(* Logix 5000 project; controller Turck_IOLink_All_Full_AOIs_V0_1 vendor 1 type 14 code 176 rev 32.11; software revision 32.00; part 3 of 7 *)
(* tags used below, declared in another part *)
   TBEN_I_DATA : INT[173];   // Input Data from IO Block
   TBEN_O_DATA : INT[131];   // Output Data to IO Block
   TBEN_C_DATA : SINT[160];
   DXP1_OUT : BOOL;
   DXP3_OUT : BOOL;
   DXP5_OUT : BOOL;
   DXP7_OUT : BOOL;
   IOLDevice_PORT1 : BOOL;
   IOLDevice_PORT2 : BOOL;
   IOLDevice_PORT3 : BOOL;
   IOLDevice_PORT4 : BOOL;
   IOLDevice_PORT5 : BOOL;
   IOLDevice_PORT6 : BOOL;
   IOLDevice_PORT7 : BOOL;
   IOLDevice_PORT8 : BOOL;
   DXP7_IN : BOOL;
   IOL8_DI : BOOL;
   IOL10_DI : BOOL;
   IOL12_DI : BOOL;
   IOL14_DI : BOOL;
   PORT1_Mode_IOL_or_DI : BOOL;   // 0: IO-LINK without validation 1: Port is set to DI (Power Cycle or Module Inhibit cycle require)
   PORT2_Mode_IOL_or_DI : BOOL;   // 0: IO-LINK without validation 1: Port is set to DI (Power Cycle or Module Inhibit cycle require)
   PORT3_Mode_IOL_or_DI : BOOL;   // 0: IO-LINK without validation 1: Port is set to DI (Power Cycle or Module Inhibit cycle require)
   PORT4_Mode_IOL_or_DI : BOOL;   // 0: IO-LINK without validation 1: Port is set to DI (Power Cycle or Module Inhibit cycle require)
   PORT5_Mode_IOL_or_DI : BOOL;   // 0: IO-LINK without validation 1: Port is set to DI (Power Cycle or Module Inhibit cycle require)
   PORT6_Mode_IOL_or_DI : BOOL;   // 0: IO-LINK without validation 1: Port is set to DI (Power Cycle or Module Inhibit cycle require)
   PORT7_Mode_IOL_or_DI : BOOL;   // 0: IO-LINK without validation 1: Port is set to DI (Power Cycle or Module Inhibit cycle require)
   PORT8_Mode_IOL_or_DI : BOOL;   // 0: IO-LINK without validation 1: Port is set to DI (Power Cycle or Module Inhibit cycle require)
   DisableOutput_DXP1 : BOOL;
   DisableOutput_DXP3 : BOOL;
   DisableOutput_DXP5 : BOOL;
   DisableOutput_DXP7 : BOOL;
   IOLReadActive : BOOL;
   IOLWriteActive : BOOL;
   IOL_READ_Request : BOOL;
   IOL_WRITE_Request : BOOL;
(* TBEN_Lx_8IOL_AOI, continued *)

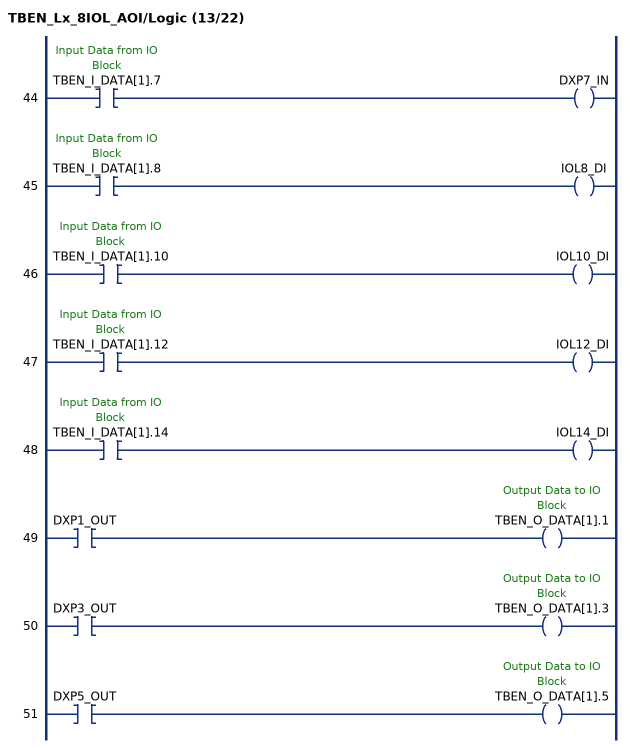
   44: XIC(TBEN_I_DATA[1].7)OTE(DXP7_IN);
   45: XIC(TBEN_I_DATA[1].8)OTE(IOL8_DI);
   46: XIC(TBEN_I_DATA[1].10)OTE(IOL10_DI);
   47: XIC(TBEN_I_DATA[1].12)OTE(IOL12_DI);
   48: XIC(TBEN_I_DATA[1].14)OTE(IOL14_DI);
   49: XIC(DXP1_OUT)OTE(TBEN_O_DATA[1].1);
   50: XIC(DXP3_OUT)OTE(TBEN_O_DATA[1].3);
   51: XIC(DXP5_OUT)OTE(TBEN_O_DATA[1].5);
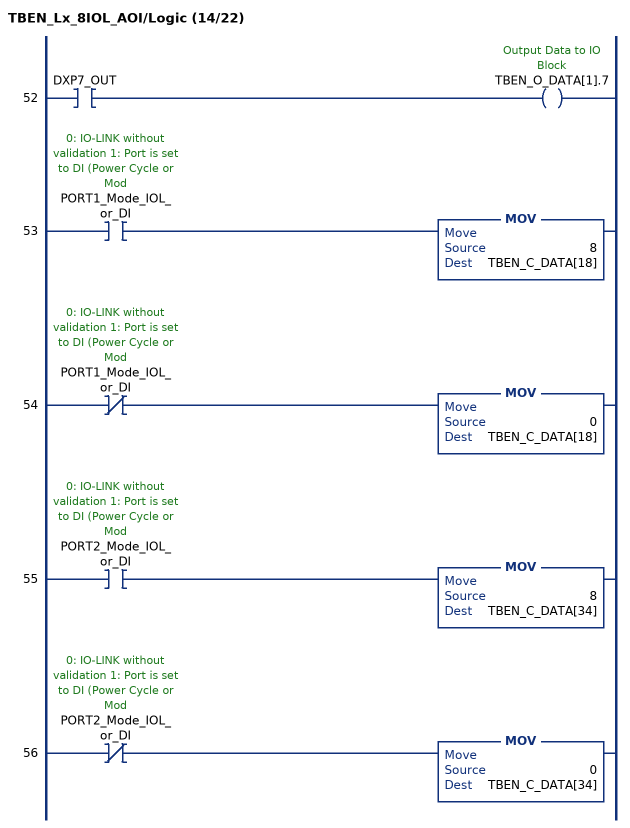
   52: XIC(DXP7_OUT)OTE(TBEN_O_DATA[1].7);
   53: XIC(PORT1_Mode_IOL_or_DI)MOV(8,TBEN_C_DATA[18]);
   54: XIO(PORT1_Mode_IOL_or_DI)MOV(0,TBEN_C_DATA[18]);
   55: XIC(PORT2_Mode_IOL_or_DI)MOV(8,TBEN_C_DATA[34]);
   56: XIO(PORT2_Mode_IOL_or_DI)MOV(0,TBEN_C_DATA[34]);
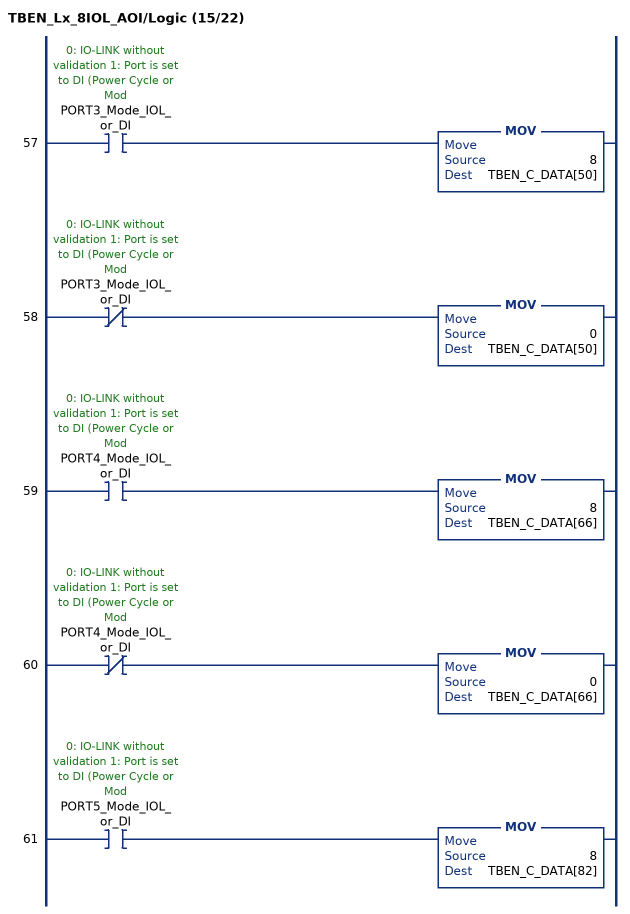
   57: XIC(PORT3_Mode_IOL_or_DI)MOV(8,TBEN_C_DATA[50]);
   58: XIO(PORT3_Mode_IOL_or_DI)MOV(0,TBEN_C_DATA[50]);
   59: XIC(PORT4_Mode_IOL_or_DI)MOV(8,TBEN_C_DATA[66]);
   60: XIO(PORT4_Mode_IOL_or_DI)MOV(0,TBEN_C_DATA[66]);
   61: XIC(PORT5_Mode_IOL_or_DI)MOV(8,TBEN_C_DATA[82]);
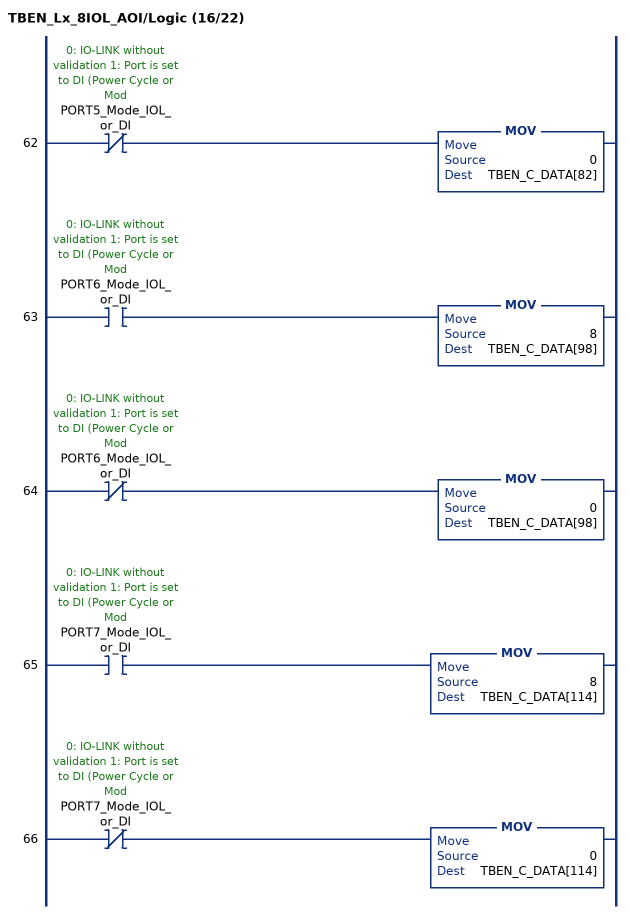
   62: XIO(PORT5_Mode_IOL_or_DI)MOV(0,TBEN_C_DATA[82]);
   63: XIC(PORT6_Mode_IOL_or_DI)MOV(8,TBEN_C_DATA[98]);
   64: XIO(PORT6_Mode_IOL_or_DI)MOV(0,TBEN_C_DATA[98]);
   65: XIC(PORT7_Mode_IOL_or_DI)MOV(8,TBEN_C_DATA[114]);
   66: XIO(PORT7_Mode_IOL_or_DI)MOV(0,TBEN_C_DATA[114]);
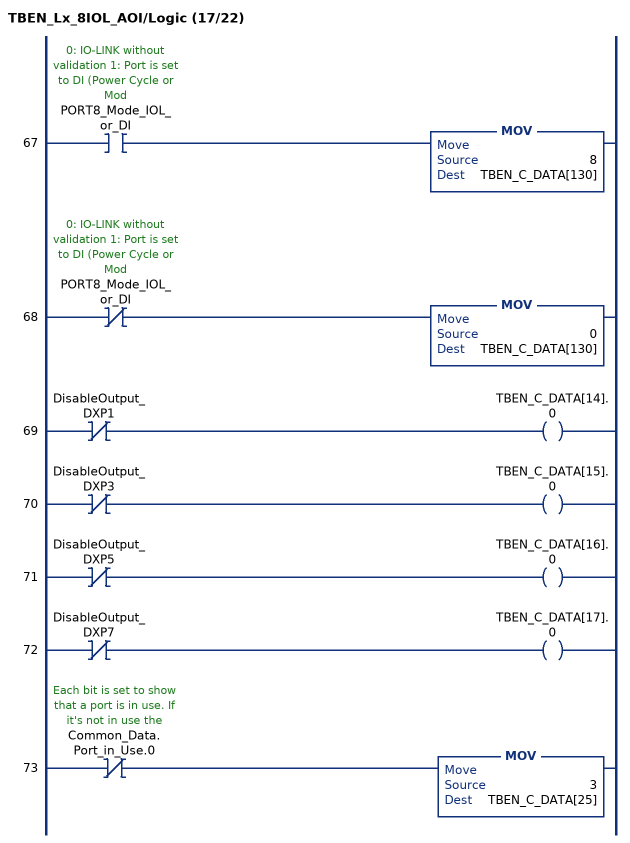
   67: XIC(PORT8_Mode_IOL_or_DI)MOV(8,TBEN_C_DATA[130]);
   68: XIO(PORT8_Mode_IOL_or_DI)MOV(0,TBEN_C_DATA[130]);
   69: XIO(DisableOutput_DXP1)OTE(TBEN_C_DATA[14].0);
   70: XIO(DisableOutput_DXP3)OTE(TBEN_C_DATA[15].0);
   71: XIO(DisableOutput_DXP5)OTE(TBEN_C_DATA[16].0);
   72: XIO(DisableOutput_DXP7)OTE(TBEN_C_DATA[17].0);
   73: XIO(Common_Data.Port_in_Use.0)MOV(3,TBEN_C_DATA[25]);
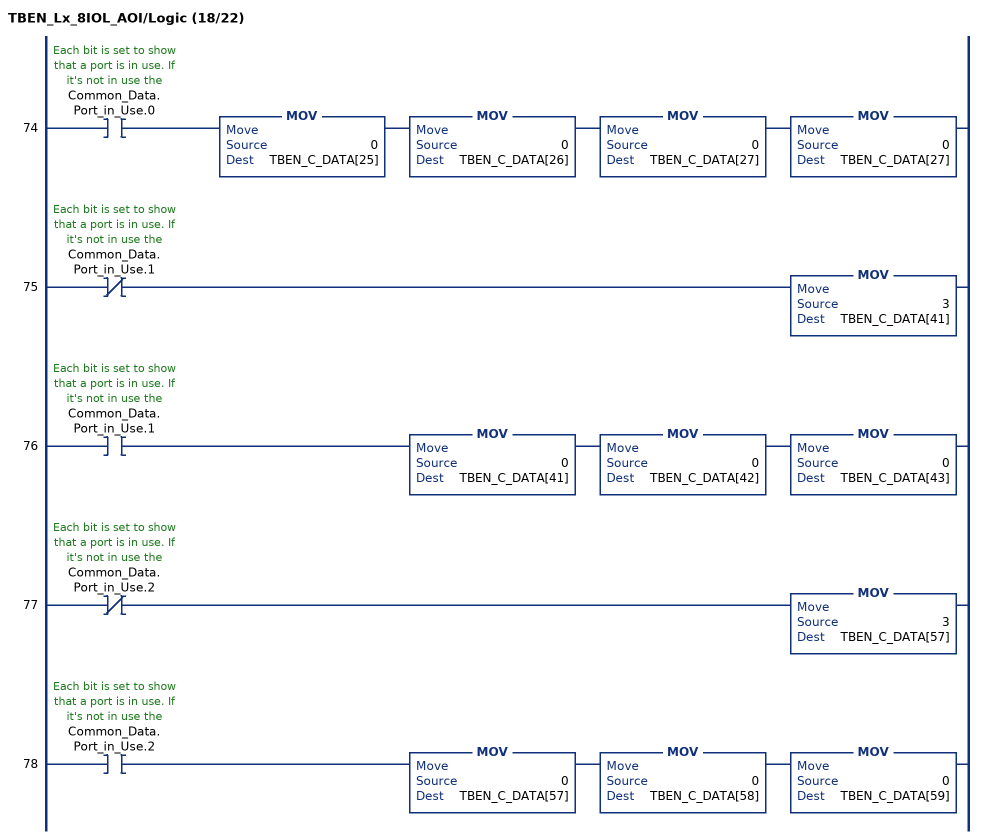
   74: XIC(Common_Data.Port_in_Use.0)MOV(0,TBEN_C_DATA[25])MOV(0,TBEN_C_DATA[26])MOV(0,TBEN_C_DATA[27])MOV(0,TBEN_C_DATA[27]);
   75: XIO(Common_Data.Port_in_Use.1)MOV(3,TBEN_C_DATA[41]);
   76: XIC(Common_Data.Port_in_Use.1)MOV(0,TBEN_C_DATA[41])MOV(0,TBEN_C_DATA[42])MOV(0,TBEN_C_DATA[43]);
   77: XIO(Common_Data.Port_in_Use.2)MOV(3,TBEN_C_DATA[57]);
   78: XIC(Common_Data.Port_in_Use.2)MOV(0,TBEN_C_DATA[57])MOV(0,TBEN_C_DATA[58])MOV(0,TBEN_C_DATA[59]);
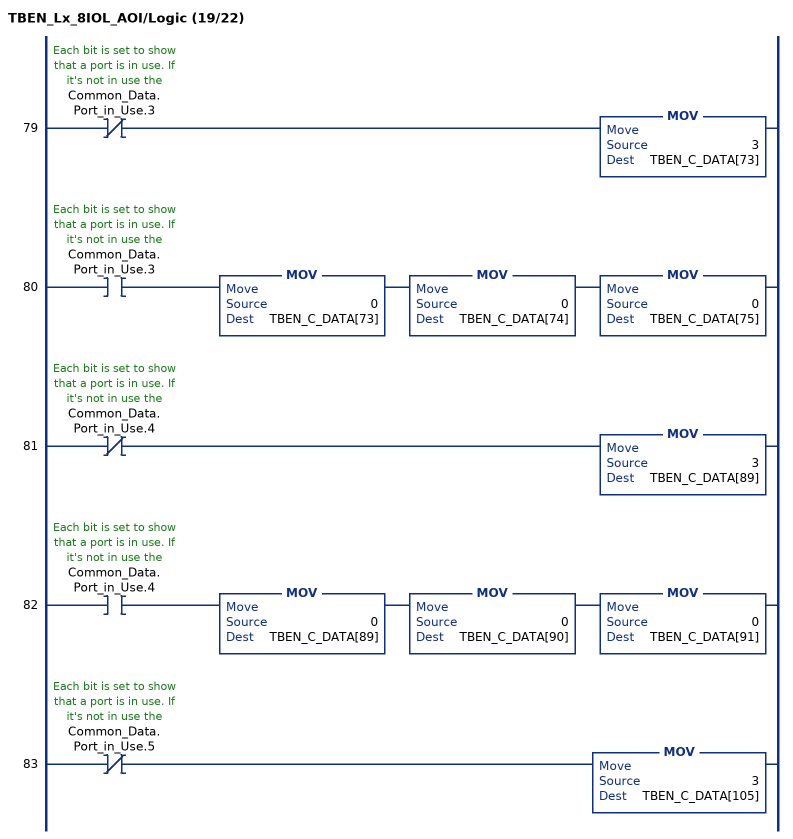
   79: XIO(Common_Data.Port_in_Use.3)MOV(3,TBEN_C_DATA[73]);
   80: XIC(Common_Data.Port_in_Use.3)MOV(0,TBEN_C_DATA[73])MOV(0,TBEN_C_DATA[74])MOV(0,TBEN_C_DATA[75]);
   81: XIO(Common_Data.Port_in_Use.4)MOV(3,TBEN_C_DATA[89]);
   82: XIC(Common_Data.Port_in_Use.4)MOV(0,TBEN_C_DATA[89])MOV(0,TBEN_C_DATA[90])MOV(0,TBEN_C_DATA[91]);
   83: XIO(Common_Data.Port_in_Use.5)MOV(3,TBEN_C_DATA[105]);
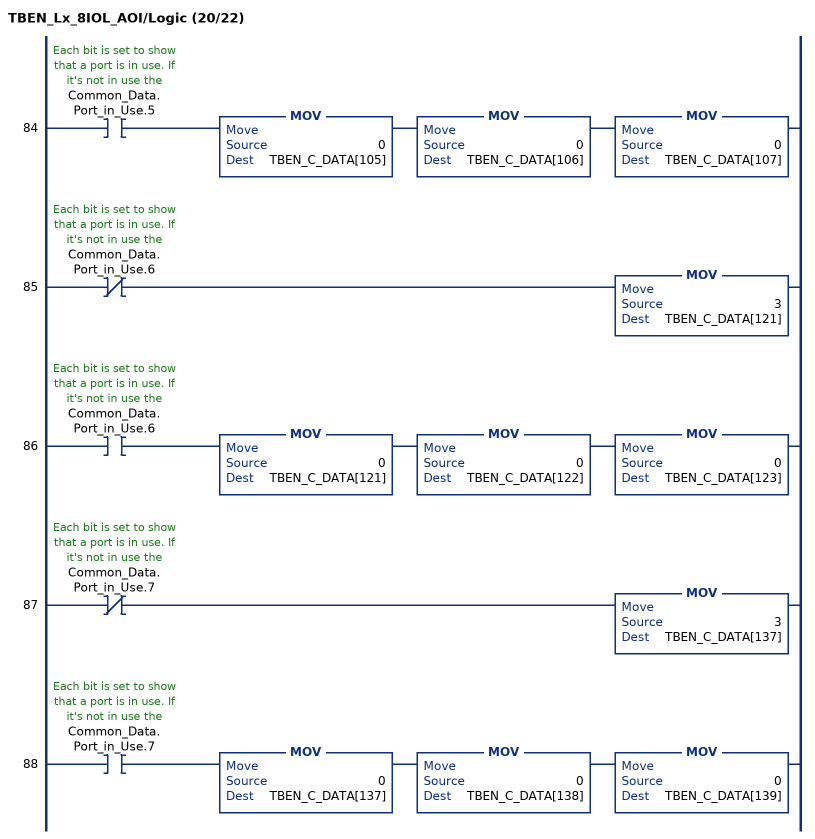
   84: XIC(Common_Data.Port_in_Use.5)MOV(0,TBEN_C_DATA[105])MOV(0,TBEN_C_DATA[106])MOV(0,TBEN_C_DATA[107]);
   85: XIO(Common_Data.Port_in_Use.6)MOV(3,TBEN_C_DATA[121]);
   86: XIC(Common_Data.Port_in_Use.6)MOV(0,TBEN_C_DATA[121])MOV(0,TBEN_C_DATA[122])MOV(0,TBEN_C_DATA[123]);
   87: XIO(Common_Data.Port_in_Use.7)MOV(3,TBEN_C_DATA[137]);
   88: XIC(Common_Data.Port_in_Use.7)MOV(0,TBEN_C_DATA[137])MOV(0,TBEN_C_DATA[138])MOV(0,TBEN_C_DATA[139]);
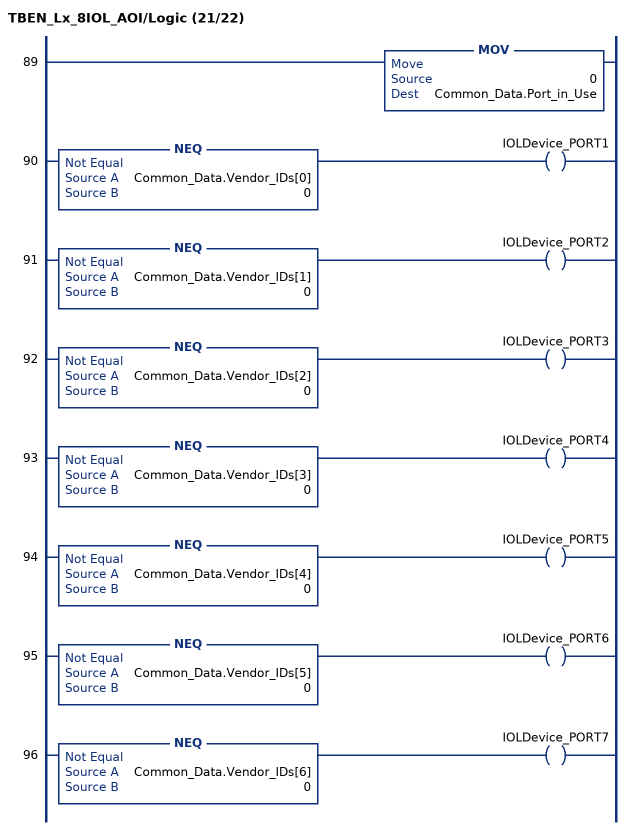
   89: MOV(0,Common_Data.Port_in_Use);
   90: NEQ(Common_Data.Vendor_IDs[0],0)OTE(IOLDevice_PORT1);
   91: NEQ(Common_Data.Vendor_IDs[1],0)OTE(IOLDevice_PORT2);
   92: NEQ(Common_Data.Vendor_IDs[2],0)OTE(IOLDevice_PORT3);
   93: NEQ(Common_Data.Vendor_IDs[3],0)OTE(IOLDevice_PORT4);
   94: NEQ(Common_Data.Vendor_IDs[4],0)OTE(IOLDevice_PORT5);
   95: NEQ(Common_Data.Vendor_IDs[5],0)OTE(IOLDevice_PORT6);
   96: NEQ(Common_Data.Vendor_IDs[6],0)OTE(IOLDevice_PORT7);
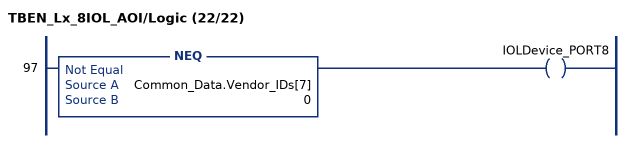
   97: NEQ(Common_Data.Vendor_IDs[7],0)OTE(IOLDevice_PORT8);
END_ROUTINE

ROUTINE Prescan   (* ladder *)
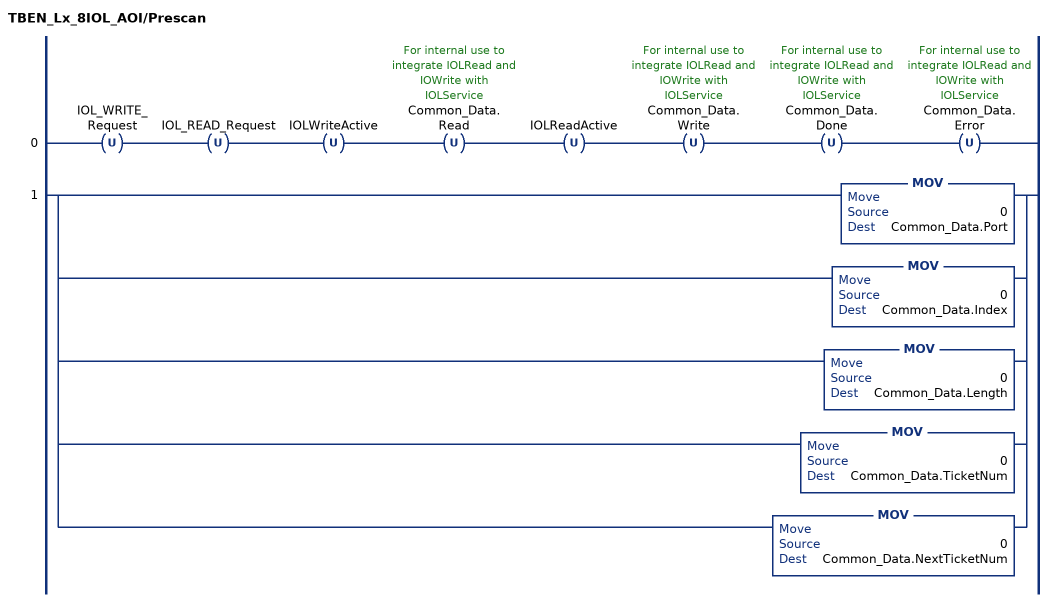
   0: OTU(IOL_WRITE_Request)OTU(IOL_READ_Request)OTU(IOLWriteActive)OTU(Common_Data.Read)OTU(IOLReadActive)OTU(Common_Data.Write)OTU(Common_Data.Done)OTU(Common_Data.Error);
   1: [MOV(0,Common_Data.Port) ,MOV(0,Common_Data.Index) ,MOV(0,Common_Data.Length) ,MOV(0,Common_Data.TicketNum) ,MOV(0,Common_Data.NextTicketNum) ];
END_ROUTINE
END_ADD_ON_INSTRUCTION

ADD_ON_INSTRUCTION Turck_IOL_Generic_AOI   (* revision 1.0 *)
VAR_INPUT
   Port : INT; {required}
END_VAR
VAR_IN_OUT
   Common_Data : Turck_IOLink_Common_Data; {required}
END_VAR
VAR_OUTPUT
   Input_Data_Word0 : INT; {visible}
   Input_Data_Word1 : INT; {visible}
   Input_Data_Word2 : INT; {visible}
   Input_Data_Word3 : INT; {visible}
   Input_Data_Word4 : INT; {visible}
   Input_Data_Word5 : INT; {visible}
   Input_Data_Word6 : INT; {visible}
   Input_Data_Word7 : INT; {visible}
   Input_Data_Word8 : INT;
   Input_Data_Word9 : INT;
   Input_Data_Word10 : INT;
   Input_Data_Word11 : INT;
   Input_Data_Word12 : INT;
   Input_Data_Word13 : INT;
   Input_Data_Word14 : INT;
   Input_Data_Word15 : INT;
END_VAR
VAR_INPUT
   Output_Data_Word0 : INT; {visible}
   Output_Data_Word1 : INT; {visible}
   Output_Data_Word2 : INT; {visible}
   Output_Data_Word3 : INT; {visible}
   Output_Data_Word4 : INT; {visible}
   Output_Data_Word5 : INT; {visible}
   Output_Data_Word6 : INT; {visible}
   Output_Data_Word7 : INT; {visible}
   Output_Data_Word8 : INT;
   Output_Data_Word9 : INT;
   Output_Data_Word10 : INT;
   Output_Data_Word11 : INT;
   Output_Data_Word12 : INT;
   Output_Data_Word13 : INT;
   Output_Data_Word14 : INT;
   Output_Data_Word15 : INT;
END_VAR
VAR
   Port_Less_One : INT; {access None}
   One : SINT; {access None}
   Port_Bit : SINT; {access None}
   Two : DINT; {access None}
END_VAR

ROUTINE Logic   (* ladder *)
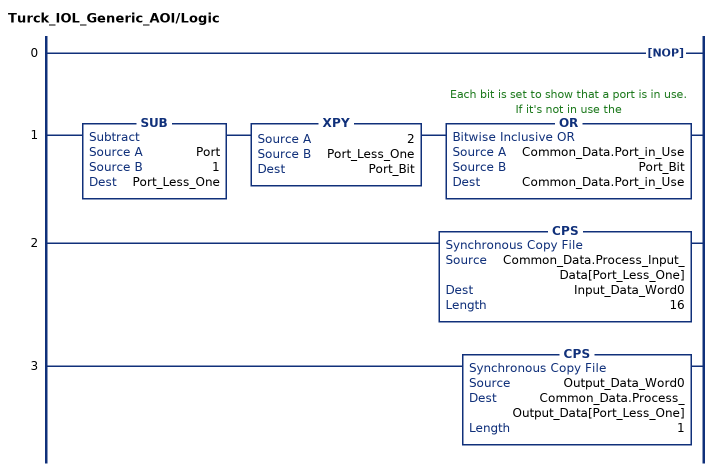
   0: NOP();
   1: SUB(Port,1,Port_Less_One)XPY(2,Port_Less_One,Port_Bit)OR(Common_Data.Port_in_Use,Port_Bit,Common_Data.Port_in_Use);
   2: CPS(Common_Data.Process_Input_Data[Port_Less_One],Input_Data_Word0,16);
   3: CPS(Output_Data_Word0,Common_Data.Process_Output_Data[Port_Less_One],1);
END_ROUTINE
END_ADD_ON_INSTRUCTION

ADD_ON_INSTRUCTION Turck_PS510_10V_Full   (* revision 1.0 *)
VAR_INPUT
   Port : INT; {required}
END_VAR
VAR_IN_OUT
   Common_Data : Turck_IOLink_Common_Data; {required}   // Controller Tag of Process Data
END_VAR
VAR_INPUT
   Units : SINT; {visible}   // Index 0x54 Subindex 1 - Change the Displayed Unit 0 = bar 1 = psi 2 = kPa 3 = MPa 4-14 = See Manual
   Menu_Lock : SINT;   // Index 0x58 - Subindex 1 - Menu Lock 0 = Unlocked 1 = Display Parameters Only 2 = Locked
   Rotate_Display : SINT; {visible}   // Index 0x5B - Subindex 1 - Display Rotation 0 = 0degrees 1 = 180 degrees
END_VAR
VAR_OUTPUT
   Pressure_PSI : REAL; {visible}
   Pressure_Bar : REAL; {visible}
   Under_Permissible : BOOL; {visible}   // Value below permissible range
   Under_Tolerance : BOOL; {visible}   // Value below tolerance range but within permissible range
   Under_Measuring : BOOL; {visible}   // Value below measuring range but within tolerance
   Over_Measuring : BOOL; {visible}   // Value above measuring range but within tolerance
   Over_Tolerance : BOOL; {visible}   // Value above tolerance range but within permissible range
   Over_Permissible : BOOL; {visible}   // Value above permissible range
   Error : BOOL; {visible}
   Process_Error : BOOL; {visible}
   EEPROM_Error : BOOL; {visible}
   Switching_State_A1 : BOOL; {visible}
   Switching_State_A2 : BOOL; {visible}
   Wrong_or_Missing_Device : BOOL; {access Read Only, visible}
END_VAR
VAR
   Measured_Value : DINT; {access None}
   Done : DINT; {access None}
   Error_DINT : DINT; {access None}
   Pending : DINT; {access None}
   Pending_or_Active : DINT; {access None}
   Port_Bit : SINT; {access None}
   Port_Less_One : SINT; {access None}
   Units_Prev : SINT; {access None}
   Output_2_Function : SINT; {access None}
   StartupCount : DINT; {access None}
   StartupDone : BOOL; {access None}
   Active : DINT; {access None}
   Read_ONS : DINT; {access None}
   MyTicketNum : INT[32]; {access None}
   Write : DINT; {access None}
   Write_ONS : DINT; {access None}
   WriteRequest : DINT; {access None}
   DoneCount : DINT; {access None}
   Status : DINT; {access None}
   ErrorCount : DINT; {access None}
   ReadRequest : DINT; {access None}
   Rotate_Display_Prev : SINT; {access None}
   Process_Data_Profile : SINT; {access None}
   Max_Pressure_Recorded_Raw : INT; {access None}
   Every_Min_Poll_TON : TIMER := (PRE := 60000); {access None}
   Min_Recorded_Pressure_Raw : INT; {access None}
   Process_Data_In_Swapped : INT; {access None}
END_VAR

ROUTINE Logic   (* ladder *)
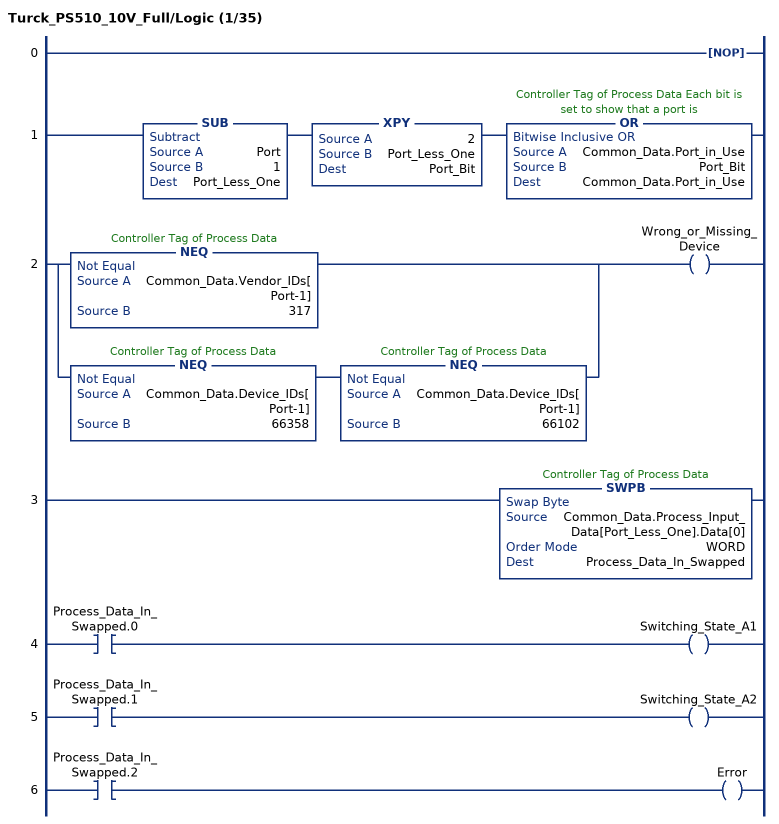
   0: NOP();
   1: SUB(Port,1,Port_Less_One)XPY(2,Port_Less_One,Port_Bit)OR(Common_Data.Port_in_Use,Port_Bit,Common_Data.Port_in_Use);
   2: [NEQ(Common_Data.Vendor_IDs[Port-1],317) ,NEQ(Common_Data.Device_IDs[Port-1],66358) NEQ(Common_Data.Device_IDs[Port-1],66102) ]OTE(Wrong_or_Missing_Device);
   3: SWPB(Common_Data.Process_Input_Data[Port_Less_One].Data[0],WORD,Process_Data_In_Swapped);
   4: XIC(Process_Data_In_Swapped.0)OTE(Switching_State_A1);
   5: XIC(Process_Data_In_Swapped.1)OTE(Switching_State_A2);
   6: XIC(Process_Data_In_Swapped.2)OTE(Error);
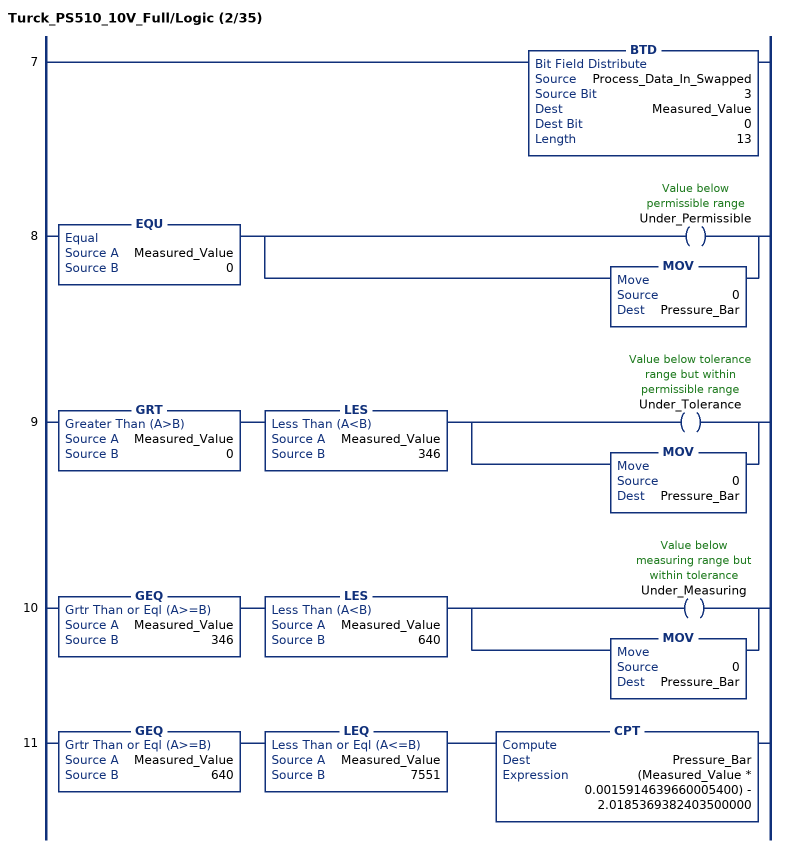
   7: BTD(Process_Data_In_Swapped,3,Measured_Value,0,13);
   8: EQU(Measured_Value,0)[OTE(Under_Permissible) ,MOV(0,Pressure_Bar) ];
   9: GRT(Measured_Value,0)LES(Measured_Value,346)[OTE(Under_Tolerance) ,MOV(0,Pressure_Bar) ];
   10: GEQ(Measured_Value,346)LES(Measured_Value,640)[OTE(Under_Measuring) ,MOV(0,Pressure_Bar) ];
   11: GEQ(Measured_Value,640)LEQ(Measured_Value,7551)CPT(Pressure_Bar,(Measured_Value * 0.0015914639660005400) - 2.0185369382403500000);
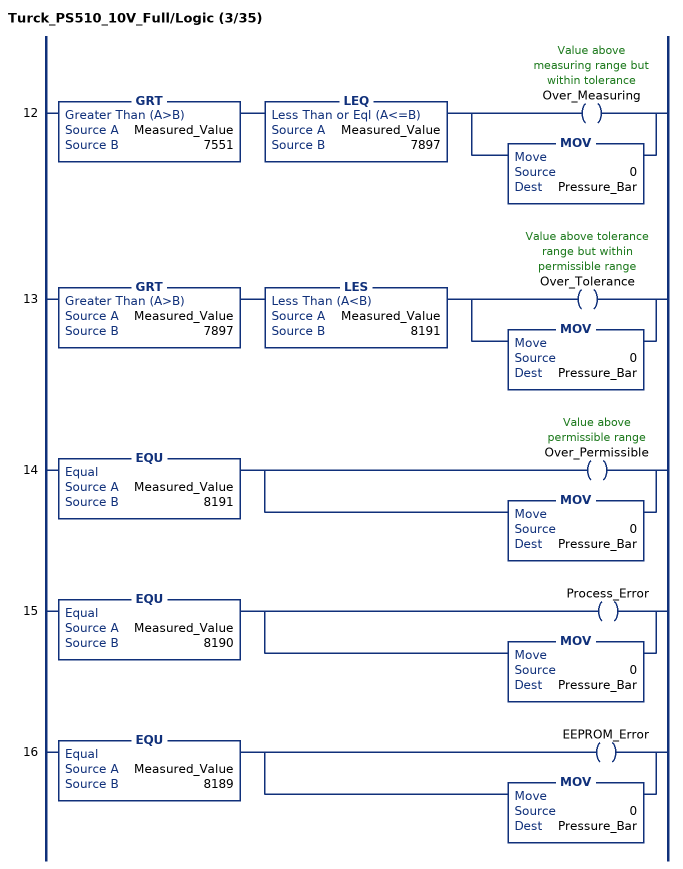
   12: GRT(Measured_Value,7551)LEQ(Measured_Value,7897)[OTE(Over_Measuring) ,MOV(0,Pressure_Bar) ];
   13: GRT(Measured_Value,7897)LES(Measured_Value,8191)[OTE(Over_Tolerance) ,MOV(0,Pressure_Bar) ];
   14: EQU(Measured_Value,8191)[OTE(Over_Permissible) ,MOV(0,Pressure_Bar) ];
   15: EQU(Measured_Value,8190)[OTE(Process_Error) ,MOV(0,Pressure_Bar) ];
   16: EQU(Measured_Value,8189)[OTE(EEPROM_Error) ,MOV(0,Pressure_Bar) ];
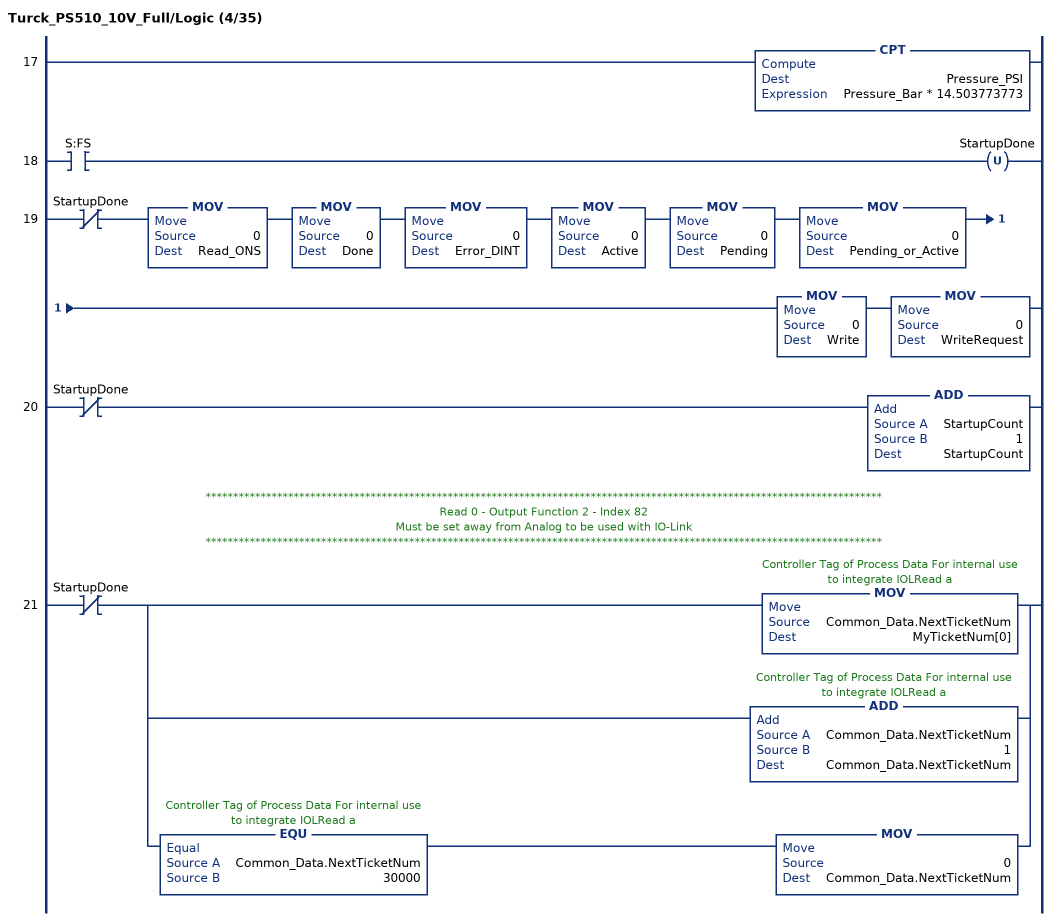
   17: CPT(Pressure_PSI,Pressure_Bar * 14.503773773);
   18: XIC(S:FS)OTU(StartupDone);
   19: XIO(StartupDone)MOV(0,Read_ONS)MOV(0,Done)MOV(0,Error_DINT)MOV(0,Active)MOV(0,Pending)MOV(0,Pending_or_Active)MOV(0,Write)MOV(0,WriteRequest);
   20: XIO(StartupDone)ADD(StartupCount,1,StartupCount);
   // ***************************************************************************************************************************
   // Read 0 - Output Function 2 - Index 82
   // Must be set away from Analog to be used with IO-Link
   // ***************************************************************************************************************************
   21: XIO(StartupDone)[MOV(Common_Data.NextTicketNum,MyTicketNum[0]) ,ADD(Common_Data.NextTicketNum,1,Common_Data.NextTicketNum) ,EQU(Common_Data.NextTicketNum,30000) MOV(0,Common_Data.NextTicketNum) ];
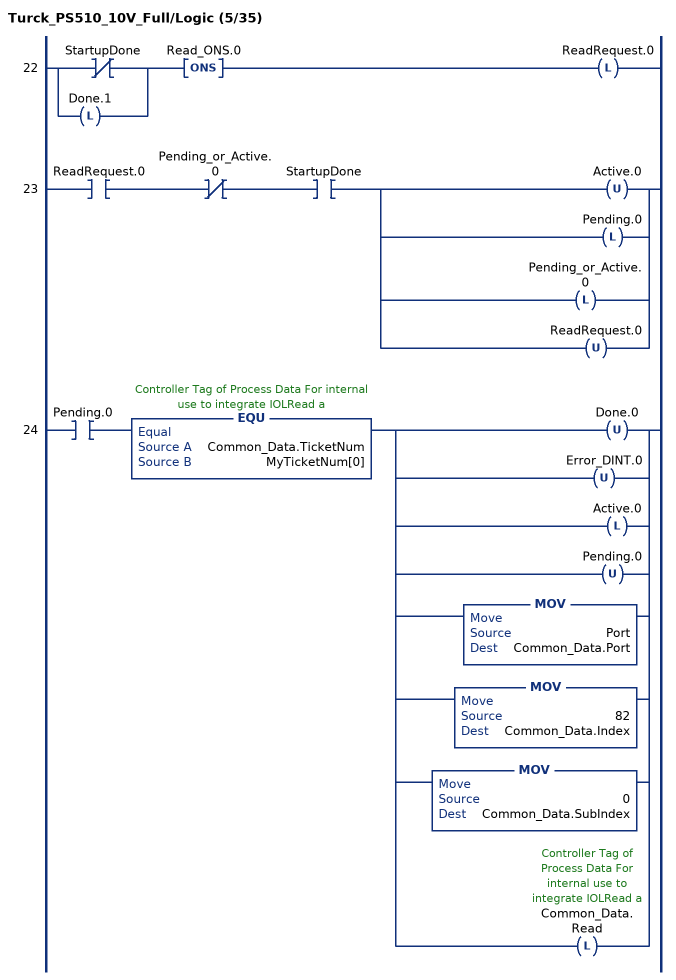
   22: [XIO(StartupDone) ,OTL(Done.1) ]ONS(Read_ONS.0)OTL(ReadRequest.0);
   23: XIC(ReadRequest.0)XIO(Pending_or_Active.0)XIC(StartupDone)[OTU(Active.0) ,OTL(Pending.0) ,OTL(Pending_or_Active.0) ,OTU(ReadRequest.0) ];
   24: XIC(Pending.0)EQU(Common_Data.TicketNum,MyTicketNum[0])[OTU(Done.0) ,OTU(Error_DINT.0) ,OTL(Active.0) ,OTU(Pending.0) ,MOV(Port,Common_Data.Port) ,MOV(82,Common_Data.Index) ,MOV(0,Common_Data.SubIndex) ,OTL(Common_Data.Read) ];
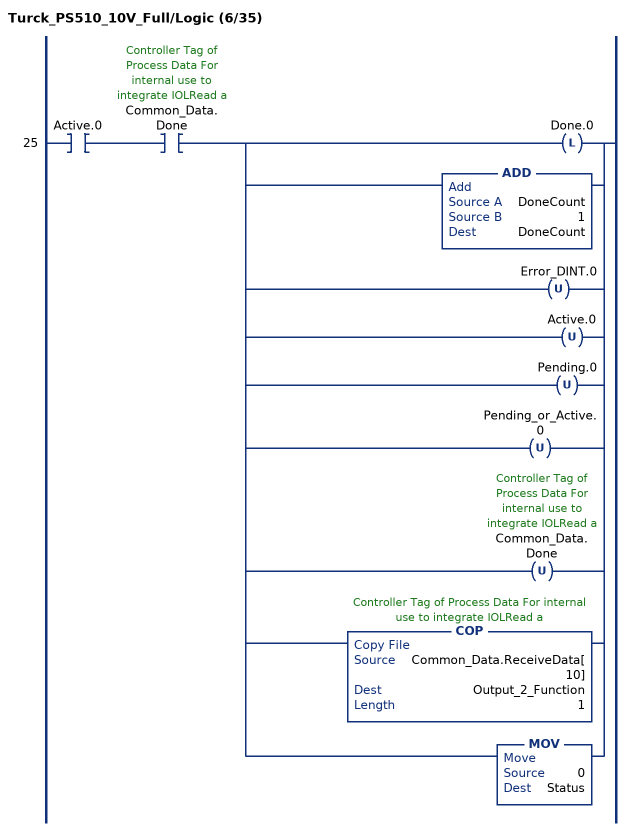
   25: XIC(Active.0)XIC(Common_Data.Done)[OTL(Done.0) ,ADD(DoneCount,1,DoneCount) ,OTU(Error_DINT.0) ,OTU(Active.0) ,OTU(Pending.0) ,OTU(Pending_or_Active.0) ,OTU(Common_Data.Done) ,COP(Common_Data.ReceiveData[10],Output_2_Function,1) ,MOV(0,Status) ];
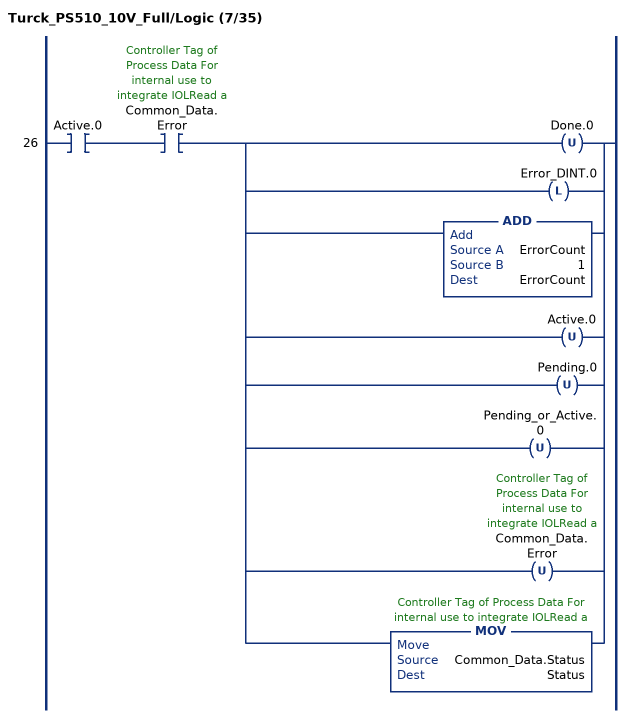
   26: XIC(Active.0)XIC(Common_Data.Error)[OTU(Done.0) ,OTL(Error_DINT.0) ,ADD(ErrorCount,1,ErrorCount) ,OTU(Active.0) ,OTU(Pending.0) ,OTU(Pending_or_Active.0) ,OTU(Common_Data.Error) ,MOV(Common_Data.Status,Status) ];
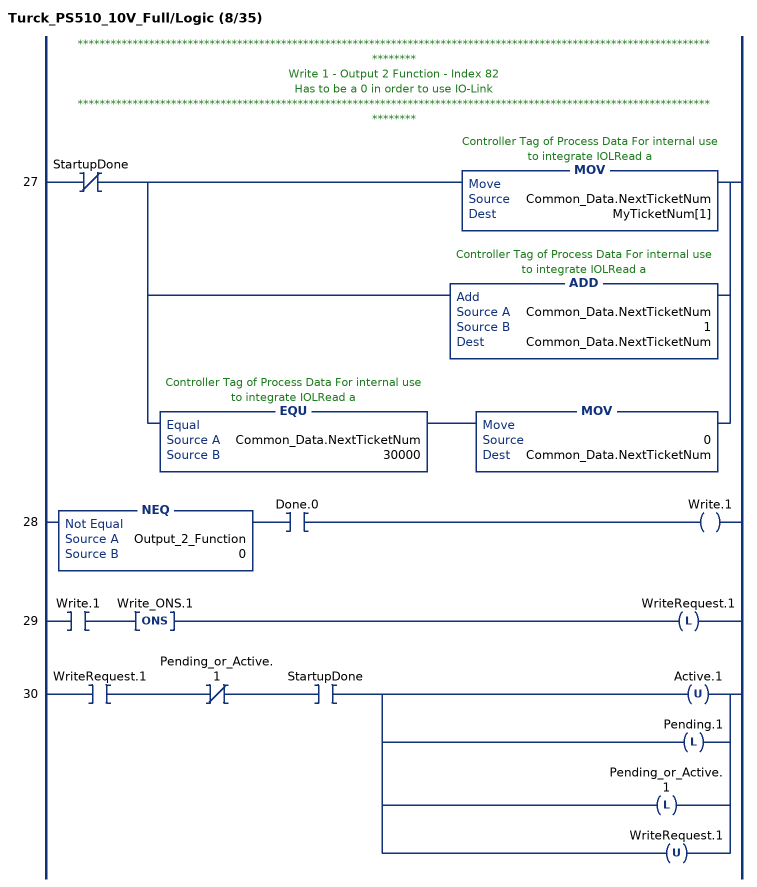
   // ***************************************************************************************************************************
   // Write 1 - Output 2 Function - Index 82
   // Has to be a 0 in order to use IO-Link
   // ***************************************************************************************************************************
   27: XIO(StartupDone)[MOV(Common_Data.NextTicketNum,MyTicketNum[1]) ,ADD(Common_Data.NextTicketNum,1,Common_Data.NextTicketNum) ,EQU(Common_Data.NextTicketNum,30000) MOV(0,Common_Data.NextTicketNum) ];
   28: NEQ(Output_2_Function,0)XIC(Done.0)OTE(Write.1);
   29: XIC(Write.1)ONS(Write_ONS.1)OTL(WriteRequest.1);
   30: XIC(WriteRequest.1)XIO(Pending_or_Active.1)XIC(StartupDone)[OTU(Active.1) ,OTL(Pending.1) ,OTL(Pending_or_Active.1) ,OTU(WriteRequest.1) ];
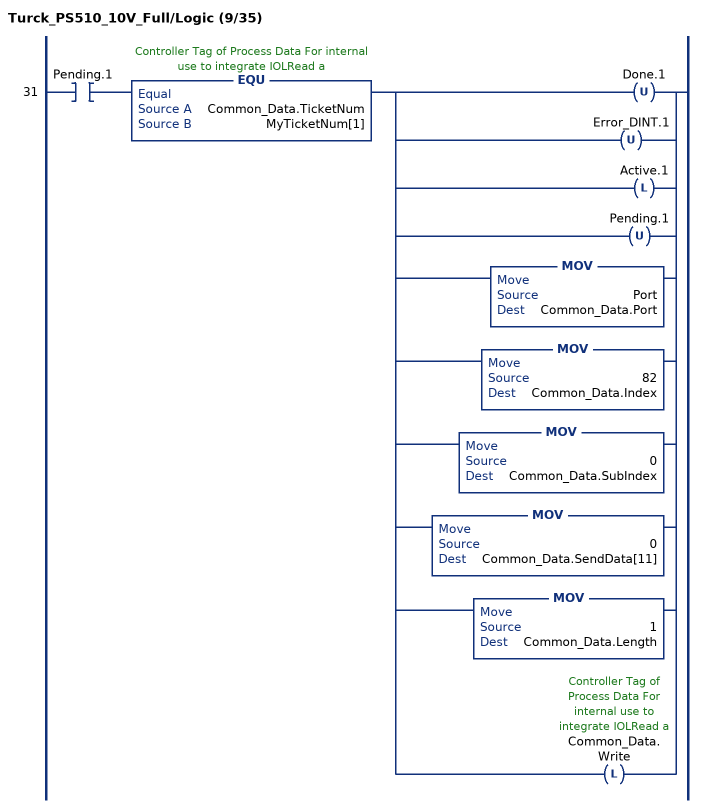
   31: XIC(Pending.1)EQU(Common_Data.TicketNum,MyTicketNum[1])[OTU(Done.1) ,OTU(Error_DINT.1) ,OTL(Active.1) ,OTU(Pending.1) ,MOV(Port,Common_Data.Port) ,MOV(82,Common_Data.Index) ,MOV(0,Common_Data.SubIndex) ,MOV(0,Common_Data.SendData[11]) ,MOV(1,Common_Data.Length) ,OTL(Common_Data.Write) ];
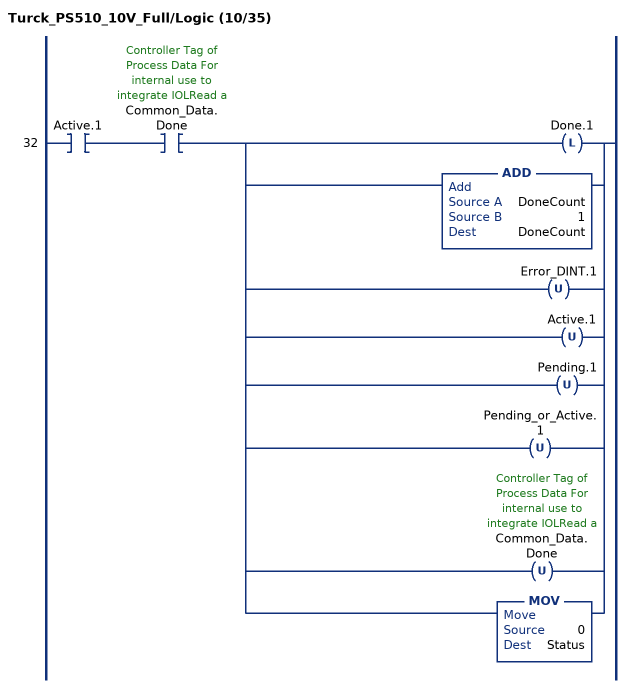
   32: XIC(Active.1)XIC(Common_Data.Done)[OTL(Done.1) ,ADD(DoneCount,1,DoneCount) ,OTU(Error_DINT.1) ,OTU(Active.1) ,OTU(Pending.1) ,OTU(Pending_or_Active.1) ,OTU(Common_Data.Done) ,MOV(0,Status) ];
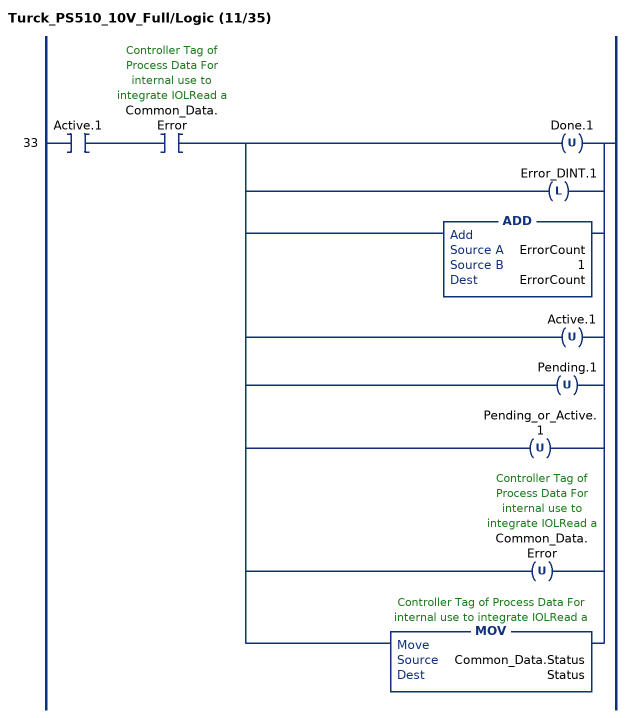
   33: XIC(Active.1)XIC(Common_Data.Error)[OTU(Done.1) ,OTL(Error_DINT.1) ,ADD(ErrorCount,1,ErrorCount) ,OTU(Active.1) ,OTU(Pending.1) ,OTU(Pending_or_Active.1) ,OTU(Common_Data.Error) ,MOV(Common_Data.Status,Status) ];
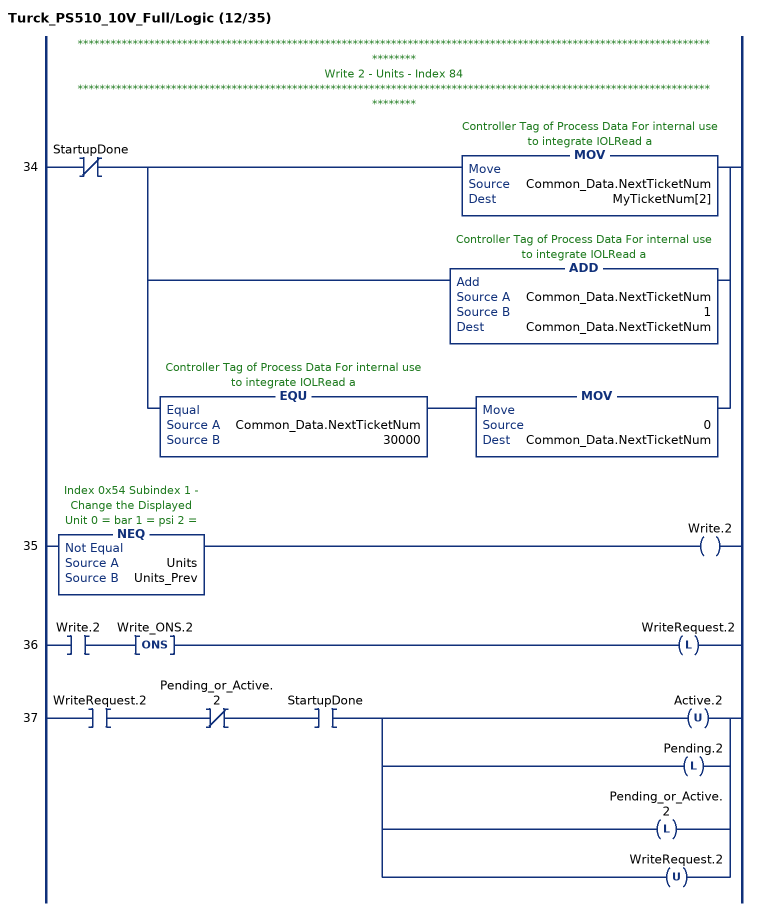
   // ***************************************************************************************************************************
   // Write 2 - Units - Index 84
   // ***************************************************************************************************************************
   34: XIO(StartupDone)[MOV(Common_Data.NextTicketNum,MyTicketNum[2]) ,ADD(Common_Data.NextTicketNum,1,Common_Data.NextTicketNum) ,EQU(Common_Data.NextTicketNum,30000) MOV(0,Common_Data.NextTicketNum) ];
   35: NEQ(Units,Units_Prev)OTE(Write.2);
   36: XIC(Write.2)ONS(Write_ONS.2)OTL(WriteRequest.2);
   37: XIC(WriteRequest.2)XIO(Pending_or_Active.2)XIC(StartupDone)[OTU(Active.2) ,OTL(Pending.2) ,OTL(Pending_or_Active.2) ,OTU(WriteRequest.2) ];
